// TIA Portal V19 export
DATA_BLOCK "UP_CM02.GP05"   // DB1005
// stored: AutoNumber false, InstanceOfName UP_Saeure.GP0x, InstanceOfType FB
"UP_Saeure.GP0x"
   // VAR RETAIN
   //    In { ExternalAccessible := 'False'; ExternalVisible := 'False'; ExternalWritable := 'False'} : Struct
   //       NotHalt : Bool;
   //       ext_Freigabe : Bool;
   //       TW_senkt : Bool;
   //       Auto : Bool;
   //       Ein : Bool;
   //       Quitt_Al_Dfl : Bool;
   //       FU_betriebsbereit : Bool;
   //       FU_Stoerung : Bool;
   //       Niv_TLS : Bool;
   //       Niv_min : Bool;
   //       Niv_max : Bool;
   //       Niv_Uel : Bool;
   //       Frg_Niv_CM05 : Bool;
   //       SRM_Saugseite_auf : Bool;
   //       SRM_Saugseite_zu : Bool;
   //       SRM_Druckseite_auf : Bool;
   //       SRM_Druckseite_zu : Bool;
   //       SRM_Eingang_Spülltg_auf : Bool;
   //       SRM_Eingang_Spülltg_zu : Bool;
   //       SRM_Ausgang_Spülltg_auf : Bool;
   //       SRM_Ausgang_Spülltg_zu : Bool;
   //       SRM_Entsogung_UV02_auf : Bool;
   //       SRM_Entsogung_UV02_zu : Bool;
   //       SRM_UV02_GP01_auf : Bool;
   //       SRM_UV02_GP01_zu : Bool;
   //       SRM_UV02_GP02_auf : Bool;
   //       SRM_UV02_GP02_zu : Bool;
   //       "SRM_GP02.QM41_auf" : Bool;
   //       "SRM_GP01.QM14_auf" : Bool;
   //       Anf_HF_Ents_CM0x : Bool;
   //       GW_p_UP : Bool;
   //       GW_LF_UP : Bool;
   //       Imp_Dfl : Bool;
   //       GW_Dfl : Bool;
   //       Tuer_zu_Seite_GP01 : Bool;
   //       Tuer_zu_vorn_GP01 : Bool;
   //       Tuer_zu_vorn_GP02 : Bool;
   //       Leckage_Doppelrohr_ok_BL26 : Bool;
   //       Leckage_Doppelschlauch_ok_BL33 : Bool;
   //       Leckage_Uml_Tunnel_ok_BL34 : Bool;
   //       Leckage_PFA_Uebergang_ok_BL16 : Bool;
   //       Leckage_PFA_Uebergang_ok_BL25 : Bool;
   //       Betriebsart : USInt;
   //       FU_speed : Int;
   //       Druck_Pumpe : Real;
   //    END_STRUCT;
   //    Param { ExternalAccessible := 'False'; ExternalVisible := 'False'; ExternalWritable := 'False'} : Struct
   //       SW_Hand : Int;
   //       SW_Auto_AZ : Int;
   //       SW_Auto_aAZ : Int;
   //       Spülzeit : Time;
   //       DT_Druckaufbau : Time;
   //       DT_Testzeit : Time;
   //       SW_Drucktest : Real;
   //       "Name" : String[12];
   //    END_STRUCT;
   //    Zst { ExternalAccessible := 'False'; ExternalVisible := 'False'; ExternalWritable := 'False'} : Struct
   //       Niveau : USInt;
   //       Status_GP0x : USInt;
   //       Status_DT : USInt;
   //       Restzeit_Spülen : Time;
   //       Restzeit_DT : Time;
   //       Spuelen : Bool;
   //       Spuelen_aktiv : Bool;
   //       Drucktest_aktiv : Bool;
   //       Umwaelzen : Bool;
   //       Weg_frei : Bool;
   //       Zeit_laeuft : Bool;
   //       Drucktest_ok : Bool;
   //       Bedienung_erlaubt : Bool;
   //       speed : Int;
   //    END_STRUCT;
   //    Mld { ExternalAccessible := 'False'; ExternalVisible := 'False'; ExternalWritable := 'False'} : Struct
   //       Niv_TLS : Bool;
   //       Niv_Ueberlauf : Bool;
   //       Niv_Sensorfehler : Bool;
   //       GW_p_UP : Bool;
   //       GW_LF_UP : Bool;
   //       GW_Dfl : Bool;
   //       UeW_Dfl_Ents : Bool;
   //       FU_nicht_bereit : Bool;
   //       FU_Stoerung : Bool;
   //       n_Auto : Bool;
   //       TO_Druckaufbau : Bool;
   //       Drucktest_ok : Bool;
   //       DT_Fehler : Bool;
   //       Pu_Spuelen_Fertig : Bool;
   //    END_STRUCT;
   //    Out { ExternalAccessible := 'False'; ExternalVisible := 'False'; ExternalWritable := 'False'} : Struct
   //       GP0x_Ein : Bool;
   //       Ventil_Saugseite : Bool;
   //       Ventil_Druckseite : Bool;
   //       Spülventil_Eingang : Bool;
   //       Spülventil_Ausgang : Bool;
   //       Entsorgung_UV02 : Bool;
   //       Ventil_UV02_GP01 : Bool;
   //       Ventil_UV02_GP02 : Bool;
   //       Soll_speed : Int;
   //    END_STRUCT;
   // END_VAR
   // VAR
   //    IEC_Timer { ExternalAccessible := 'False'; ExternalVisible := 'False'; ExternalWritable := 'False'} : Struct
   //       Spülen { S7_SetPoint := 'True'} : TP_TIME;
   //       GW_p { S7_SetPoint := 'True'} : TON_TIME;
   //       GW_Dfl { S7_SetPoint := 'True'} : TON_TIME;
   //       Imp_Dfl { S7_SetPoint := 'True'} : TON_TIME;
   //       Drucktest { S7_SetPoint := 'True'} : TP_TIME;
   //       TO_Druckaufbau { S7_SetPoint := 'True'} : TON_TIME;
   //       Spülventil_Ausgang { S7_SetPoint := 'True'} : TOF_TIME;
   //    END_STRUCT;
   //    R_TRIG_Hand_EIN { ExternalAccessible := 'False'; ExternalVisible := 'False'; ExternalWritable := 'False'} : R_TRIG;
   // END_VAR
BEGIN
END_DATA_BLOCK
